# EPICS autosave request: ADApp/Db/NDFileJPEG_settings.req
$(P)$(R)JPEGQuality
file "NDPluginFile_settings.req", P=$(P), R=$(R)
